// TIA Portal V20 export
TYPE "typeAxisInterlock"
// stored: Access Published
   STRUCT
      permit : "typeAxisInterlockpermit";
      source : "typeAxisInterlockSource";
   END_STRUCT;
END_TYPE
